	                                        //Beschränkung mögliche Nummer in der Zeile 5
	                                        FOR #i := 36 TO 44 BY 1 DO
	                                            IF #gitter[#k].nummer > 0 THEN
	                                                #gitter[#i].potenz_nummer[#gitter[#k].nummer - 1] := FALSE;
	                                            END_IF;
	                                        END_FOR;
	                                        //Beschränkung mögliche Nummer in der Säule 6
	                                        FOR #i := 5 TO 80 BY 9 DO
	                                            IF #gitter[#k].nummer > 0 THEN
	                                                #gitter[#i].potenz_nummer[#gitter[#k].nummer - 1] := FALSE;
	                                            END_IF;
	                                        END_FOR;
	                                        //Beschränkung mögliche Nummer in dem Viereck 5
	                                        #initial := 30;
	                                        #länge := 32;
	                                        FOR #m := 0 TO 2 BY 1 DO
	                                            FOR #i := #initial TO #länge BY 1 DO
	                                                IF #gitter[#k].nummer > 0 THEN
	                                                    #gitter[#i].potenz_nummer[#gitter[#k].nummer - 1] := FALSE;
	                                                END_IF;
	                                            END_FOR;
	                                            IF #m < 2 THEN
	                                                #initial := #initial + 9;
	                                                #länge := #länge + 9;
	                                            END_IF;
	                                        END_FOR;
	                                    END_REGION
	                                    //Feldchen 43
	                                42:
	                                    REGION Feldchen 43
	                                        //Beschränkung mögliche Nummer in der Zeile 5
	                                        FOR #i := 36 TO 44 BY 1 DO
	                                            IF #gitter[#k].nummer > 0 THEN
	                                                #gitter[#i].potenz_nummer[#gitter[#k].nummer - 1] := FALSE;
	                                            END_IF;
	                                        END_FOR;
	                                        //Beschränkung mögliche Nummer in der Säule 7
	                                        FOR #i := 6 TO 80 BY 9 DO
	                                            IF #gitter[#k].nummer > 0 THEN
	                                                #gitter[#i].potenz_nummer[#gitter[#k].nummer - 1] := FALSE;
	                                            END_IF;
	                                        END_FOR;
	                                        //Beschränkung mögliche Nummer in dem Viereck 6
	                                        #initial := 33;
	                                        #länge := 35;
	                                        FOR #m := 0 TO 2 BY 1 DO
	                                            FOR #i := #initial TO #länge BY 1 DO
	                                                IF #gitter[#k].nummer > 0 THEN
	                                                    #gitter[#i].potenz_nummer[#gitter[#k].nummer - 1] := FALSE;
	                                                END_IF;
	                                            END_FOR;
	                                            IF #m < 2 THEN
	                                                #initial := #initial + 9;
	                                                #länge := #länge + 9;
	                                            END_IF;
	                                        END_FOR;
	                                    END_REGION
	                                    //Feldchen 44
	                                43:
	                                    REGION Feldchen 44
	                                        //Beschränkung mögliche Nummer in der Zeile 5
	                                        FOR #i := 36 TO 44 BY 1 DO
	                                            IF #gitter[#k].nummer > 0 THEN
	                                                #gitter[#i].potenz_nummer[#gitter[#k].nummer - 1] := FALSE;
	                                            END_IF;
	                                        END_FOR;
	                                        //Beschränkung mögliche Nummer in der Säule 8
	                                        FOR #i := 7 TO 80 BY 9 DO
	                                            IF #gitter[#k].nummer > 0 THEN
	                                                #gitter[#i].potenz_nummer[#gitter[#k].nummer - 1] := FALSE;
	                                            END_IF;
	                                        END_FOR;
	                                        //Beschränkung mögliche Nummer in dem Viereck 6
	                                        #initial := 33;
	                                        #länge := 35;
	                                        FOR #m := 0 TO 2 BY 1 DO
	                                            FOR #i := #initial TO #länge BY 1 DO
	                                                IF #gitter[#k].nummer > 0 THEN
	                                                    #gitter[#i].potenz_nummer[#gitter[#k].nummer - 1] := FALSE;
	                                                END_IF;
	                                            END_FOR;
	                                            IF #m < 2 THEN
	                                                #initial := #initial + 9;
	                                                #länge := #länge + 9;
	                                            END_IF;
	                                        END_FOR;
	                                    END_REGION
	                                    //Feldchen 45
	                                44:
	                                    REGION Feldchen 45
	                                        //Beschränkung mögliche Nummer in der Zeile 5
	                                        FOR #i := 36 TO 44 BY 1 DO
	                                            IF #gitter[#k].nummer > 0 THEN
	                                                #gitter[#i].potenz_nummer[#gitter[#k].nummer - 1] := FALSE;
	                                            END_IF;
	                                        END_FOR;
	                                        //Beschränkung mögliche Nummer in der Säule 9
	                                        FOR #i := 8 TO 80 BY 9 DO
	                                            IF #gitter[#k].nummer > 0 THEN
	                                                #gitter[#i].potenz_nummer[#gitter[#k].nummer - 1] := FALSE;
	                                            END_IF;
	                                        END_FOR;
	                                        //Beschränkung mögliche Nummer in dem Viereck 6
	                                        #initial := 33;
	                                        #länge := 35;
	                                        FOR #m := 0 TO 2 BY 1 DO
	                                            FOR #i := #initial TO #länge BY 1 DO
	                                                IF #gitter[#k].nummer > 0 THEN
	                                                    #gitter[#i].potenz_nummer[#gitter[#k].nummer - 1] := FALSE;
	                                                END_IF;
	                                            END_FOR;
	                                            IF #m < 2 THEN
	                                                #initial := #initial + 9;
	                                                #länge := #länge + 9;
	                                            END_IF;
	                                        END_FOR;
	                                    END_REGION
	                                    //Feldchen 46
	                                45:
	                                    REGION Feldchen 46
	                                        //Beschränkung mögliche Nummer in der Zeile 6
	                                        FOR #i := 45 TO 53 BY 1 DO
	                                            IF #gitter[#k].nummer > 0 THEN
	                                                #gitter[#i].potenz_nummer[#gitter[#k].nummer - 1] := FALSE;
	                                            END_IF;
	                                        END_FOR;
	                                        //Beschränkung mögliche Nummer in der Säule 1
	                                        FOR #i := 0 TO 80 BY 9 DO
	                                            IF #gitter[#k].nummer > 0 THEN
	                                                #gitter[#i].potenz_nummer[#gitter[#k].nummer - 1] := FALSE;
	                                            END_IF;
	                                        END_FOR;
	                                        //Beschränkung mögliche Nummer in dem Viereck 4
	                                        #initial := 27;
	                                        #länge := 29;
	                                        FOR #m := 0 TO 2 BY 1 DO
	                                            FOR #i := #initial TO #länge BY 1 DO
	                                                IF #gitter[#k].nummer > 0 THEN
	                                                    #gitter[#i].potenz_nummer[#gitter[#k].nummer - 1] := FALSE;
	                                                END_IF;
	                                            END_FOR;
	                                            IF #m < 2 THEN
	                                                #initial := #initial + 9;
	                                                #länge := #länge + 9;
	                                            END_IF;
	                                        END_FOR;
	                                    END_REGION
	                                    //Feldchen 47
	                                46:
	                                    REGION Feldchen 47
	                                        //Beschränkung mögliche Nummer in der Zeile 6
	                                        FOR #i := 45 TO 53 BY 1 DO
	                                            IF #gitter[#k].nummer > 0 THEN
	                                                #gitter[#i].potenz_nummer[#gitter[#k].nummer - 1] := FALSE;
	                                            END_IF;
	                                        END_FOR;
	                                        //Beschränkung mögliche Nummer in der Säule 2
	                                        FOR #i := 1 TO 80 BY 9 DO
	                                            IF #gitter[#k].nummer > 0 THEN
	                                                #gitter[#i].potenz_nummer[#gitter[#k].nummer - 1] := FALSE;
	                                            END_IF;
	                                        END_FOR;
	                                        //Beschränkung mögliche Nummer in dem Viereck 4
	                                        #initial := 27;
	                                        #länge := 29;
	                                        FOR #m := 0 TO 2 BY 1 DO
	                                            FOR #i := #initial TO #länge BY 1 DO
	                                                IF #gitter[#k].nummer > 0 THEN
	                                                    #gitter[#i].potenz_nummer[#gitter[#k].nummer - 1] := FALSE;
	                                                END_IF;
	                                            END_FOR;
	                                            IF #m < 2 THEN
	                                                #initial := #initial + 9;
	                                                #länge := #länge + 9;
	                                            END_IF;
	                                        END_FOR;
	                                    END_REGION
	                                    //Feldchen 48
	                                47:
	                                    REGION Feldchen 48
	                                        //Beschränkung mögliche Nummer in der Zeile 6
	                                        FOR #i := 45 TO 53 BY 1 DO
	                                            IF #gitter[#k].nummer > 0 THEN
	                                                #gitter[#i].potenz_nummer[#gitter[#k].nummer - 1] := FALSE;
	                                            END_IF;
	                                        END_FOR;
	                                        //Beschränkung mögliche Nummer in der Säule 3
	                                        FOR #i := 2 TO 80 BY 9 DO
	                                            IF #gitter[#k].nummer > 0 THEN
	                                                #gitter[#i].potenz_nummer[#gitter[#k].nummer - 1] := FALSE;
	                                            END_IF;
	                                        END_FOR;
	                                        //Beschränkung mögliche Nummer in dem Viereck 4
	                                        #initial := 27;
	                                        #länge := 29;
	                                        FOR #m := 0 TO 2 BY 1 DO
	                                            FOR #i := #initial TO #länge BY 1 DO
	                                                IF #gitter[#k].nummer > 0 THEN
	                                                    #gitter[#i].potenz_nummer[#gitter[#k].nummer - 1] := FALSE;
	                                                END_IF;
	                                            END_FOR;
	                                            IF #m < 2 THEN
	                                                #initial := #initial + 9;
	                                                #länge := #länge + 9;
	                                            END_IF;
	                                        END_FOR;
	                                    END_REGION
	                                    //Feldchen 49
	                                48:
	                                    REGION Feldchen 49
	                                        //Beschränkung mögliche Nummer in der Zeile 6
	                                        FOR #i := 45 TO 53 BY 1 DO
	                                            IF #gitter[#k].nummer > 0 THEN
	                                                #gitter[#i].potenz_nummer[#gitter[#k].nummer - 1] := FALSE;
	                                            END_IF;
	                                        END_FOR;
	                                        //Beschränkung mögliche Nummer in der Säule 4
	                                        FOR #i := 3 TO 80 BY 9 DO
	                                            IF #gitter[#k].nummer > 0 THEN
	                                                #gitter[#i].potenz_nummer[#gitter[#k].nummer - 1] := FALSE;
	                                            END_IF;
	                                        END_FOR;
	                                        //Beschränkung mögliche Nummer in dem Viereck 5
	                                        #initial := 30;
	                                        #länge := 32;
	                                        FOR #m := 0 TO 2 BY 1 DO
	                                            FOR #i := #initial TO #länge BY 1 DO
	                                                IF #gitter[#k].nummer > 0 THEN
	                                                    #gitter[#i].potenz_nummer[#gitter[#k].nummer - 1] := FALSE;
	                                                END_IF;
	                                            END_FOR;
	                                            IF #m < 2 THEN
	                                                #initial := #initial + 9;
	                                                #länge := #länge + 9;
	                                            END_IF;
	                                        END_FOR;
	                                    END_REGION
	                                    //Feldchen 50
	                                49:
	                                    REGION Feldchen 50
	                                        //Beschränkung mögliche Nummer in der Zeile 6
	                                        FOR #i := 45 TO 53 BY 1 DO
	                                            IF #gitter[#k].nummer > 0 THEN
	                                                #gitter[#i].potenz_nummer[#gitter[#k].nummer - 1] := FALSE;
	                                            END_IF;
	                                        END_FOR;
	                                        //Beschränkung mögliche Nummer in der Säule 5
	                                        FOR #i := 4 TO 80 BY 9 DO
	                                            IF #gitter[#k].nummer > 0 THEN
	                                                #gitter[#i].potenz_nummer[#gitter[#k].nummer - 1] := FALSE;
	                                            END_IF;
	                                        END_FOR;
	                                        //Beschränkung mögliche Nummer in dem Viereck 5
	                                        #initial := 30;
	                                        #länge := 32;
	                                        FOR #m := 0 TO 2 BY 1 DO
	                                            FOR #i := #initial TO #länge BY 1 DO
	                                                IF #gitter[#k].nummer > 0 THEN
	                                                    #gitter[#i].potenz_nummer[#gitter[#k].nummer - 1] := FALSE;
	                                                END_IF;
	                                            END_FOR;
	                                            IF #m < 2 THEN
	                                                #initial := #initial + 9;
	                                                #länge := #länge + 9;
	                                            END_IF;
	                                        END_FOR;
	                                    END_REGION
	                                    //Feldchen 51
	                                50:
	                                    REGION Feldchen 51
	                                        //Beschränkung mögliche Nummer in der Zeile 6
	                                        FOR #i := 45 TO 53 BY 1 DO
	                                            IF #gitter[#k].nummer > 0 THEN
	                                                #gitter[#i].potenz_nummer[#gitter[#k].nummer - 1] := FALSE;
	                                            END_IF;
	                                        END_FOR;
	                                        //Beschränkung mögliche Nummer in der Säule 6
	                                        FOR #i := 5 TO 80 BY 9 DO
	                                            IF #gitter[#k].nummer > 0 THEN
	                                                #gitter[#i].potenz_nummer[#gitter[#k].nummer - 1] := FALSE;
	                                            END_IF;
	                                        END_FOR;
	                                        //Beschränkung mögliche Nummer in dem Viereck 5
	                                        #initial := 30;
	                                        #länge := 32;
	                                        FOR #m := 0 TO 2 BY 1 DO
	                                            FOR #i := #initial TO #länge BY 1 DO
	                                                IF #gitter[#k].nummer > 0 THEN
	                                                    #gitter[#i].potenz_nummer[#gitter[#k].nummer - 1] := FALSE;
	                                                END_IF;
	                                            END_FOR;
	                                            IF #m < 2 THEN
	                                                #initial := #initial + 9;
	                                                #länge := #länge + 9;
	                                            END_IF;
	                                        END_FOR;
	                                    END_REGION
	                                    //Feldchen 52
	                                51:
	                                    REGION Feldchen 52
	                                        //Beschränkung mögliche Nummer in der Zeile 6
	                                        FOR #i := 45 TO 53 BY 1 DO
	                                            IF #gitter[#k].nummer > 0 THEN
	                                                #gitter[#i].potenz_nummer[#gitter[#k].nummer - 1] := FALSE;
	                                            END_IF;
	                                        END_FOR;
	                                        //Beschränkung mögliche Nummer in der Säule 7
	                                        FOR #i := 6 TO 80 BY 9 DO
	                                            IF #gitter[#k].nummer > 0 THEN
	                                                #gitter[#i].potenz_nummer[#gitter[#k].nummer - 1] := FALSE;
	                                            END_IF;
	                                        END_FOR;
	                                        //Beschränkung mögliche Nummer in dem Viereck 6
	                                        #initial := 33;
	                                        #länge := 35;
	                                        FOR #m := 0 TO 2 BY 1 DO
	                                            FOR #i := #initial TO #länge BY 1 DO
	                                                IF #gitter[#k].nummer > 0 THEN
	                                                    #gitter[#i].potenz_nummer[#gitter[#k].nummer - 1] := FALSE;
	                                                END_IF;
	                                            END_FOR;
	                                            IF #m < 2 THEN
	                                                #initial := #initial + 9;
	                                                #länge := #länge + 9;
	                                            END_IF;
	                                        END_FOR;
	                                    END_REGION
	                                    //Feldchen 53
	                                52:
	                                    REGION Feldchen 53
	                                        //Beschränkung mögliche Nummer in der Zeile 6
	                                        FOR #i := 45 TO 53 BY 1 DO
	                                            IF #gitter[#k].nummer > 0 THEN
	                                                #gitter[#i].potenz_nummer[#gitter[#k].nummer - 1] := FALSE;
	                                            END_IF;
	                                        END_FOR;
	                                        //Beschränkung mögliche Nummer in der Säule 8
	                                        FOR #i := 7 TO 80 BY 9 DO
	                                            IF #gitter[#k].nummer > 0 THEN
	                                                #gitter[#i].potenz_nummer[#gitter[#k].nummer - 1] := FALSE;
	                                            END_IF;
	                                        END_FOR;
	                                        //Beschränkung mögliche Nummer in dem Viereck 6
	                                        #initial := 33;
	                                        #länge := 35;
	                                        FOR #m := 0 TO 2 BY 1 DO
	                                            FOR #i := #initial TO #länge BY 1 DO
	                                                IF #gitter[#k].nummer > 0 THEN
	                                                    #gitter[#i].potenz_nummer[#gitter[#k].nummer - 1] := FALSE;
	                                                END_IF;
	                                            END_FOR;
	                                            IF #m < 2 THEN
	                                                #initial := #initial + 9;
	                                                #länge := #länge + 9;
	                                            END_IF;
	                                        END_FOR;
	                                    END_REGION
	                                    //Feldchen 54
	                                53:
	                                    REGION Feldchen 54
	                                        //Beschränkung mögliche Nummer in der Zeile 6
	                                        FOR #i := 45 TO 53 BY 1 DO
	                                            IF #gitter[#k].nummer > 0 THEN
	                                                #gitter[#i].potenz_nummer[#gitter[#k].nummer - 1] := FALSE;
	                                            END_IF;
	                                        END_FOR;
	                                        //Beschränkung mögliche Nummer in der Säule 9
	                                        FOR #i := 8 TO 80 BY 9 DO
	                                            IF #gitter[#k].nummer > 0 THEN
	                                                #gitter[#i].potenz_nummer[#gitter[#k].nummer - 1] := FALSE;
	                                            END_IF;
	                                        END_FOR;
	                                        //Beschränkung mögliche Nummer in dem Viereck 6
	                                        #initial := 33;
	                                        #länge := 35;
	                                        FOR #m := 0 TO 2 BY 1 DO
	                                            FOR #i := #initial TO #länge BY 1 DO
	                                                IF #gitter[#k].nummer > 0 THEN
	                                                    #gitter[#i].potenz_nummer[#gitter[#k].nummer - 1] := FALSE;
	                                                END_IF;
	                                            END_FOR;
	                                            IF #m < 2 THEN
	                                                #initial := #initial + 9;
	                                                #länge := #länge + 9;
	                                            END_IF;
	                                        END_FOR;
	                                    END_REGION
	                                    //Feldchen 55
	                                54:
	                                    REGION Feldchen 55
	                                        //Beschränkung mögliche Nummer in der Zeile 7
	                                        FOR #i := 54 TO 62 BY 1 DO
	                                            IF #gitter[#k].nummer > 0 THEN
	                                                #gitter[#i].potenz_nummer[#gitter[#k].nummer - 1] := FALSE;
	                                            END_IF;
	                                        END_FOR;
	                                        //Beschränkung mögliche Nummer in der Säule 1
	                                        FOR #i := 0 TO 80 BY 9 DO
	                                            IF #gitter[#k].nummer > 0 THEN
	                                                #gitter[#i].potenz_nummer[#gitter[#k].nummer - 1] := FALSE;
	                                            END_IF;
	                                        END_FOR;
	                                        //Beschränkung mögliche Nummer in dem Viereck 7
	                                        #initial := 54;
	                                        #länge := 56;
	                                        FOR #m := 0 TO 2 BY 1 DO
	                                            FOR #i := #initial TO #länge BY 1 DO
	                                                IF #gitter[#k].nummer > 0 THEN
	                                                    #gitter[#i].potenz_nummer[#gitter[#k].nummer - 1] := FALSE;
	                                                END_IF;
	                                            END_FOR;
	                                            IF #m < 2 THEN
	                                                #initial := #initial + 9;
	                                                #länge := #länge + 9;
	                                            END_IF;
	                                        END_FOR;
	                                    END_REGION
	                                    //Feldchen 56
	                                55:
	                                    REGION Feldchen 56
	                                        //Beschränkung mögliche Nummer in der Zeile 7
	                                        FOR #i := 54 TO 62 BY 1 DO
	                                            IF #gitter[#k].nummer > 0 THEN
	                                                #gitter[#i].potenz_nummer[#gitter[#k].nummer - 1] := FALSE;
	                                            END_IF;
	                                        END_FOR;
	                                        //Beschränkung mögliche Nummer in der Säule 2
	                                        FOR #i := 1 TO 80 BY 9 DO
	                                            IF #gitter[#k].nummer > 0 THEN
	                                                #gitter[#i].potenz_nummer[#gitter[#k].nummer - 1] := FALSE;
	                                            END_IF;
	                                        END_FOR;
	                                        //Beschränkung mögliche Nummer in dem Viereck 7
	                                        #initial := 54;
	                                        #länge := 56;
	                                        FOR #m := 0 TO 2 BY 1 DO
	                                            FOR #i := #initial TO #länge BY 1 DO
	                                                IF #gitter[#k].nummer > 0 THEN
	                                                    #gitter[#i].potenz_nummer[#gitter[#k].nummer - 1] := FALSE;
	                                                END_IF;
	                                            END_FOR;
	                                            IF #m < 2 THEN
	                                                #initial := #initial + 9;
	                                                #länge := #länge + 9;
	                                            END_IF;
	                                        END_FOR;
	                                    END_REGION
	                                    //Feldchen 57
	                                56:
	                                    REGION Feldchen 57
	                                        //Beschränkung mögliche Nummer in der Zeile 7
	                                        FOR #i := 54 TO 62 BY 1 DO
	                                            IF #gitter[#k].nummer > 0 THEN
	                                                #gitter[#i].potenz_nummer[#gitter[#k].nummer - 1] := FALSE;
	                                            END_IF;
	                                        END_FOR;
	                                        //Beschränkung mögliche Nummer in der Säule 3
	                                        FOR #i := 2 TO 80 BY 9 DO
	                                            IF #gitter[#k].nummer > 0 THEN
	                                                #gitter[#i].potenz_nummer[#gitter[#k].nummer - 1] := FALSE;
	                                            END_IF;
	                                        END_FOR;
	                                        //Beschränkung mögliche Nummer in dem Viereck 7
	                                        #initial := 54;
	                                        #länge := 56;
	                                        FOR #m := 0 TO 2 BY 1 DO
	                                            FOR #i := #initial TO #länge BY 1 DO
	                                                IF #gitter[#k].nummer > 0 THEN
	                                                    #gitter[#i].potenz_nummer[#gitter[#k].nummer - 1] := FALSE;
	                                                END_IF;
	                                            END_FOR;
	                                            IF #m < 2 THEN
	                                                #initial := #initial + 9;
	                                                #länge := #länge + 9;
	                                            END_IF;
	                                        END_FOR;
	                                    END_REGION //Feldchen 57
	                                    //Feldchen 58
	                                57:
	                                    REGION Feldchen 58
	                                        //Beschränkung mögliche Nummer in der Zeile 7
	                                        FOR #i := 54 TO 62 BY 1 DO
	                                            IF #gitter[#k].nummer > 0 THEN
	                                                #gitter[#i].potenz_nummer[#gitter[#k].nummer - 1] := FALSE;
	                                            END_IF;
	                                        END_FOR;
	                                        //Beschränkung mögliche Nummer in der Säule 4
	                                        FOR #i := 3 TO 80 BY 9 DO
	                                            IF #gitter[#k].nummer > 0 THEN
	                                                #gitter[#i].potenz_nummer[#gitter[#k].nummer - 1] := FALSE;
	                                            END_IF;
	                                        END_FOR;
	                                        //Beschränkung mögliche Nummer in dem Viereck 8
	                                        #initial := 57;
	                                        #länge := 59;
	                                        FOR #m := 0 TO 2 BY 1 DO
	                                            FOR #i := #initial TO #länge BY 1 DO
	                                                IF #gitter[#k].nummer > 0 THEN
	                                                    #gitter[#i].potenz_nummer[#gitter[#k].nummer - 1] := FALSE;
	                                                END_IF;
	                                            END_FOR;
	                                            IF #m < 2 THEN
	                                                #initial := #initial + 9;
	                                                #länge := #länge + 9;
	                                            END_IF;
	                                        END_FOR;
	                                    END_REGION
	                                    //Feldchen 59
	                                58:
	                                    REGION Feldchen 59
	                                        //Beschränkung mögliche Nummer in der Zeile 7
	                                        FOR #i := 54 TO 62 BY 1 DO
	                                            IF #gitter[#k].nummer > 0 THEN
	                                                #gitter[#i].potenz_nummer[#gitter[#k].nummer - 1] := FALSE;
	                                            END_IF;
	                                        END_FOR;
	                                        //Beschränkung mögliche Nummer in der Säule 5
	                                        FOR #i := 4 TO 80 BY 9 DO
	                                            IF #gitter[#k].nummer > 0 THEN
	                                                #gitter[#i].potenz_nummer[#gitter[#k].nummer - 1] := FALSE;
	                                            END_IF;
	                                        END_FOR;
	                                        //Beschränkung mögliche Nummer in dem Viereck 8
	                                        #initial := 57;
	                                        #länge := 59;
	                                        FOR #m := 0 TO 2 BY 1 DO
	                                            FOR #i := #initial TO #länge BY 1 DO
	                                                IF #gitter[#k].nummer > 0 THEN
	                                                    #gitter[#i].potenz_nummer[#gitter[#k].nummer - 1] := FALSE;
	                                                END_IF;
	                                            END_FOR;
	                                            IF #m < 2 THEN
	                                                #initial := #initial + 9;
	                                                #länge := #länge + 9;
	                                            END_IF;
	                                        END_FOR;
	                                    END_REGION
	                                    //Feldchen 60
	                                59:
	                                    REGION Feldchen 60
	                                        //Beschränkung mögliche Nummer in der Zeile 7
	                                        FOR #i := 54 TO 62 BY 1 DO
	                                            IF #gitter[#k].nummer > 0 THEN
	                                                #gitter[#i].potenz_nummer[#gitter[#k].nummer - 1] := FALSE;
	                                            END_IF;
	                                        END_FOR;
	                                        //Beschränkung mögliche Nummer in der Säule 6
	                                        FOR #i := 5 TO 80 BY 9 DO
	                                            IF #gitter[#k].nummer > 0 THEN
	                                                #gitter[#i].potenz_nummer[#gitter[#k].nummer - 1] := FALSE;
	                                            END_IF;
	                                        END_FOR;
	                                        //Beschränkung mögliche Nummer in dem Viereck 8
	                                        #initial := 57;
	                                        #länge := 59;
	                                        FOR #m := 0 TO 2 BY 1 DO
	                                            FOR #i := #initial TO #länge BY 1 DO
	                                                IF #gitter[#k].nummer > 0 THEN
	                                                    #gitter[#i].potenz_nummer[#gitter[#k].nummer - 1] := FALSE;
	                                                END_IF;
	                                            END_FOR;
	                                            IF #m < 2 THEN
	                                                #initial := #initial + 9;
	                                                #länge := #länge + 9;
	                                            END_IF;
	                                        END_FOR;
	                                    END_REGION
	                                    //Feldchen 61
	                                60:
	                                    REGION Feldchen 61
	                                        //Beschränkung mögliche Nummer in der Zeile 7
	                                        FOR #i := 54 TO 62 BY 1 DO
	                                            IF #gitter[#k].nummer > 0 THEN
	                                                #gitter[#i].potenz_nummer[#gitter[#k].nummer - 1] := FALSE;
	                                            END_IF;
	                                        END_FOR;
	                                        //Beschränkung mögliche Nummer in der Säule 7
	                                        FOR #i := 6 TO 80 BY 9 DO
	                                            IF #gitter[#k].nummer > 0 THEN
	                                                #gitter[#i].potenz_nummer[#gitter[#k].nummer - 1] := FALSE;
	                                            END_IF;
	                                        END_FOR;
	                                        //Beschränkung mögliche Nummer in dem Viereck 9
	                                        #initial := 60;
	                                        #länge := 62;
	                                        FOR #m := 0 TO 2 BY 1 DO
	                                            FOR #i := #initial TO #länge BY 1 DO
	                                                IF #gitter[#k].nummer > 0 THEN
	                                                    #gitter[#i].potenz_nummer[#gitter[#k].nummer - 1] := FALSE;
	                                                END_IF;
	                                            END_FOR;
	                                            IF #m < 2 THEN
	                                                #initial := #initial + 9;
	                                                #länge := #länge + 9;
	                                            END_IF;
	                                        END_FOR;
	                                    END_REGION
	                                    //Feldchen 62
	                                61:
	                                    REGION Feldchen 62
	                                        //Beschränkung mögliche Nummer in der Zeile 7
	                                        FOR #i := 54 TO 62 BY 1 DO
	                                            IF #gitter[#k].nummer > 0 THEN
	                                                #gitter[#i].potenz_nummer[#gitter[#k].nummer - 1] := FALSE;
	                                            END_IF;
	                                        END_FOR;
	                                        //Beschränkung mögliche Nummer in der Säule 8
	                                        FOR #i := 7 TO 80 BY 9 DO
	                                            IF #gitter[#k].nummer > 0 THEN
	                                                #gitter[#i].potenz_nummer[#gitter[#k].nummer - 1] := FALSE;
	                                            END_IF;
	                                        END_FOR;
	                                        //Beschränkung mögliche Nummer in dem Viereck 9
	                                        #initial := 60;
	                                        #länge := 62;
	                                        FOR #m := 0 TO 2 BY 1 DO
	                                            FOR #i := #initial TO #länge BY 1 DO
	                                                IF #gitter[#k].nummer > 0 THEN
	                                                    #gitter[#i].potenz_nummer[#gitter[#k].nummer - 1] := FALSE;
	                                                END_IF;
	                                            END_FOR;
	                                            IF #m < 2 THEN
	                                                #initial := #initial + 9;
	                                                #länge := #länge + 9;
	                                            END_IF;
	                                        END_FOR;
	                                    END_REGION
	                                    //Feldchen 63
	                                62:
	                                    REGION Feldchen 63
	                                        //Beschränkung mögliche Nummer in der Zeile 7
	                                        FOR #i := 54 TO 62 BY 1 DO
	                                            IF #gitter[#k].nummer > 0 THEN
	                                                #gitter[#i].potenz_nummer[#gitter[#k].nummer - 1] := FALSE;
	                                            END_IF;
	                                        END_FOR;
	                                        //Beschränkung mögliche Nummer in der Säule 9
	                                        FOR #i := 8 TO 80 BY 9 DO
	                                            IF #gitter[#k].nummer > 0 THEN
	                                                #gitter[#i].potenz_nummer[#gitter[#k].nummer - 1] := FALSE;
	                                            END_IF;
	                                        END_FOR;
	                                        //Beschränkung mögliche Nummer in dem Viereck 9
	                                        #initial := 60;
	                                        #länge := 62;
	                                        FOR #m := 0 TO 2 BY 1 DO
	                                            FOR #i := #initial TO #länge BY 1 DO
	                                                IF #gitter[#k].nummer > 0 THEN
	                                                    #gitter[#i].potenz_nummer[#gitter[#k].nummer - 1] := FALSE;
	                                                END_IF;
	                                            END_FOR;
	                                            IF #m < 2 THEN
	                                                #initial := #initial + 9;
	                                                #länge := #länge + 9;
	                                            END_IF;
	                                        END_FOR;
	                                    END_REGION
	                                    //Feldchen 64
	                                63:
	                                    REGION Feldchen 64
	                                        //Beschränkung mögliche Nummer in der Zeile 8
	                                        FOR #i := 63 TO 71 BY 1 DO
	                                            IF #gitter[#k].nummer > 0 THEN
	                                                #gitter[#i].potenz_nummer[#gitter[#k].nummer - 1] := FALSE;
	                                            END_IF;
	                                        END_FOR;
	                                        //Beschränkung mögliche Nummer in der Säule 1
	                                        FOR #i := 0 TO 80 BY 9 DO
	                                            IF #gitter[#k].nummer > 0 THEN
	                                                #gitter[#i].potenz_nummer[#gitter[#k].nummer - 1] := FALSE;
	                                            END_IF;
	                                        END_FOR;
	                                        //Beschränkung mögliche Nummer in dem Viereck 7
	                                        #initial := 54;
	                                        #länge := 56;
	                                        FOR #m := 0 TO 2 BY 1 DO
	                                            FOR #i := #initial TO #länge BY 1 DO
	                                                IF #gitter[#k].nummer > 0 THEN
	                                                    #gitter[#i].potenz_nummer[#gitter[#k].nummer - 1] := FALSE;
	                                                END_IF;
	                                            END_FOR;
	                                            IF #m < 2 THEN
	                                                #initial := #initial + 9;
	                                                #länge := #länge + 9;
	                                            END_IF;
	                                        END_FOR;
	                                    END_REGION
	                                    //Feldchen 65
	                                64:
	                                    REGION Feldchen 65
	                                        //Beschränkung mögliche Nummer in der Zeile 8
	                                        FOR #i := 63 TO 71 BY 1 DO
	                                            IF #gitter[#k].nummer > 0 THEN
	                                                #gitter[#i].potenz_nummer[#gitter[#k].nummer - 1] := FALSE;
	                                            END_IF;
	                                        END_FOR;
	                                        //Beschränkung mögliche Nummer in der Säule 2
	                                        FOR #i := 1 TO 80 BY 9 DO
	                                            IF #gitter[#k].nummer > 0 THEN
	                                                #gitter[#i].potenz_nummer[#gitter[#k].nummer - 1] := FALSE;
	                                            END_IF;
	                                        END_FOR;
	                                        //Beschränkung mögliche Nummer in dem Viereck 7
	                                        #initial := 54;
	                                        #länge := 56;
	                                        FOR #m := 0 TO 2 BY 1 DO
	                                            FOR #i := #initial TO #länge BY 1 DO
	                                                IF #gitter[#k].nummer > 0 THEN
	                                                    #gitter[#i].potenz_nummer[#gitter[#k].nummer - 1] := FALSE;
	                                                END_IF;
	                                            END_FOR;
	                                            IF #m < 2 THEN
	                                                #initial := #initial + 9;
	                                                #länge := #länge + 9;
	                                            END_IF;
	                                        END_FOR;
	                                    END_REGION
	                                    //Feldchen 66
	                                65:
	                                    REGION Feldchen 66
	                                        //Beschränkung mögliche Nummer in der Zeile 8
	                                        FOR #i := 63 TO 71 BY 1 DO
	                                            IF #gitter[#k].nummer > 0 THEN
	                                                #gitter[#i].potenz_nummer[#gitter[#k].nummer - 1] := FALSE;
	                                            END_IF;
	                                        END_FOR;
	                                        //Beschränkung mögliche Nummer in der Säule 3
	                                        FOR #i := 2 TO 80 BY 9 DO
	                                            IF #gitter[#k].nummer > 0 THEN
	                                                #gitter[#i].potenz_nummer[#gitter[#k].nummer - 1] := FALSE;
	                                            END_IF;
	                                        END_FOR;
	                                        //Beschränkung mögliche Nummer in dem Viereck 7
	                                        #initial := 54;
	                                        #länge := 56;
	                                        FOR #m := 0 TO 2 BY 1 DO
	                                            FOR #i := #initial TO #länge BY 1 DO
	                                                IF #gitter[#k].nummer > 0 THEN
	                                                    #gitter[#i].potenz_nummer[#gitter[#k].nummer - 1] := FALSE;
	                                                END_IF;
	                                            END_FOR;
	                                            IF #m < 2 THEN
	                                                #initial := #initial + 9;
	                                                #länge := #länge + 9;
	                                            END_IF;
	                                        END_FOR;
	                                    END_REGION
	                                    //Feldchen 67
	                                66:
	                                    REGION Feldchen 67
	                                        //Beschränkung mögliche Nummer in der Zeile 8
	                                        FOR #i := 63 TO 71 BY 1 DO
	                                            IF #gitter[#k].nummer > 0 THEN
	                                                #gitter[#i].potenz_nummer[#gitter[#k].nummer - 1] := FALSE;
	                                            END_IF;
	                                        END_FOR;
	                                        //Beschränkung mögliche Nummer in der Säule 4
	                                        FOR #i := 3 TO 80 BY 9 DO
	                                            IF #gitter[#k].nummer > 0 THEN
	                                                #gitter[#i].potenz_nummer[#gitter[#k].nummer - 1] := FALSE;
	                                            END_IF;
	                                        END_FOR;
	                                        //Beschränkung mögliche Nummer in dem Viereck 8
	                                        #initial := 57;
	                                        #länge := 59;
	                                        FOR #m := 0 TO 2 BY 1 DO
	                                            FOR #i := #initial TO #länge BY 1 DO
	                                                IF #gitter[#k].nummer > 0 THEN
	                                                    #gitter[#i].potenz_nummer[#gitter[#k].nummer - 1] := FALSE;
	                                                END_IF;
	                                            END_FOR;
	                                            IF #m < 2 THEN
	                                                #initial := #initial + 9;
	                                                #länge := #länge + 9;
	                                            END_IF;
	                                        END_FOR;
	                                    END_REGION
	                                    //Feldchen 68
	                                67:
	                                    REGION Feldchen 68
	                                        //Beschränkung mögliche Nummer in der Zeile 8
	                                        FOR #i := 63 TO 71 BY 1 DO
	                                            IF #gitter[#k].nummer > 0 THEN
	                                                #gitter[#i].potenz_nummer[#gitter[#k].nummer - 1] := FALSE;
	                                            END_IF;
	                                        END_FOR;
	                                        //Beschränkung mögliche Nummer in der Säule 5
	                                        FOR #i := 4 TO 80 BY 9 DO
	                                            IF #gitter[#k].nummer > 0 THEN
	                                                #gitter[#i].potenz_nummer[#gitter[#k].nummer - 1] := FALSE;
	                                            END_IF;
	                                        END_FOR;
	                                        //Beschränkung mögliche Nummer in dem Viereck 8
	                                        #initial := 57;
	                                        #länge := 59;
	                                        FOR #m := 0 TO 2 BY 1 DO
	                                            FOR #i := #initial TO #länge BY 1 DO
	                                                IF #gitter[#k].nummer > 0 THEN
	                                                    #gitter[#i].potenz_nummer[#gitter[#k].nummer - 1] := FALSE;
	                                                END_IF;
	                                            END_FOR;
	                                            IF #m < 2 THEN
	                                                #initial := #initial + 9;
	                                                #länge := #länge + 9;
	                                            END_IF;
	                                        END_FOR;
	                                    END_REGION
	                                    //Feldchen 69
	                                68:
	                                    REGION Feldchen 69
	                                        //Beschränkung mögliche Nummer in der Zeile 8
	                                        FOR #i := 63 TO 71 BY 1 DO
	                                            IF #gitter[#k].nummer > 0 THEN
	                                                #gitter[#i].potenz_nummer[#gitter[#k].nummer - 1] := FALSE;
	                                            END_IF;
	                                        END_FOR;
	                                        //Beschränkung mögliche Nummer in der Säule 6
	                                        FOR #i := 5 TO 80 BY 9 DO
	                                            IF #gitter[#k].nummer > 0 THEN
	                                                #gitter[#i].potenz_nummer[#gitter[#k].nummer - 1] := FALSE;
	                                            END_IF;
	                                        END_FOR;
	                                        //Beschränkung mögliche Nummer in dem Viereck 8
	                                        #initial := 57;
	                                        #länge := 59;
	                                        FOR #m := 0 TO 2 BY 1 DO
	                                            FOR #i := #initial TO #länge BY 1 DO
	                                                IF #gitter[#k].nummer > 0 THEN
	                                                    #gitter[#i].potenz_nummer[#gitter[#k].nummer - 1] := FALSE;
	                                                END_IF;
	                                            END_FOR;
	                                            IF #m < 2 THEN
	                                                #initial := #initial + 9;
	                                                #länge := #länge + 9;
	                                            END_IF;
	                                        END_FOR;
	                                    END_REGION
	                                    //Feldchen 70
	                                69:
	                                    REGION Feldchen 70
	                                        //Beschränkung mögliche Nummer in der Zeile 8
	                                        FOR #i := 63 TO 71 BY 1 DO
	                                            IF #gitter[#k].nummer > 0 THEN
	                                                #gitter[#i].potenz_nummer[#gitter[#k].nummer - 1] := FALSE;
	                                            END_IF;
	                                        END_FOR;
	                                        //Beschränkung mögliche Nummer in der Säule 7
	                                        FOR #i := 6 TO 80 BY 9 DO
	                                            IF #gitter[#k].nummer > 0 THEN
	                                                #gitter[#i].potenz_nummer[#gitter[#k].nummer - 1] := FALSE;
	                                            END_IF;
	                                        END_FOR;
	                                        //Beschränkung mögliche Nummer in dem Viereck 9
	                                        #initial := 60;
	                                        #länge := 62;
	                                        FOR #m := 0 TO 2 BY 1 DO
	                                            FOR #i := #initial TO #länge BY 1 DO
	                                                IF #gitter[#k].nummer > 0 THEN
	                                                    #gitter[#i].potenz_nummer[#gitter[#k].nummer - 1] := FALSE;
	                                                END_IF;
	                                            END_FOR;
	                                            IF #m < 2 THEN
	                                                #initial := #initial + 9;
	                                                #länge := #länge + 9;
	                                            END_IF;
	                                        END_FOR;
	                                    END_REGION
	                                    //Feldchen 71
	                                70:
	                                    REGION Feldchen 71
	                                        //Beschränkung mögliche Nummer in der Zeile 8
	                                        FOR #i := 63 TO 71 BY 1 DO
	                                            IF #gitter[#k].nummer > 0 THEN
	                                                #gitter[#i].potenz_nummer[#gitter[#k].nummer - 1] := FALSE;
	                                            END_IF;
	                                        END_FOR;
	                                        //Beschränkung mögliche Nummer in der Säule 8
	                                        FOR #i := 7 TO 80 BY 9 DO
	                                            IF #gitter[#k].nummer > 0 THEN
	                                                #gitter[#i].potenz_nummer[#gitter[#k].nummer - 1] := FALSE;
	                                            END_IF;
	                                        END_FOR;
	                                        //Beschränkung mögliche Nummer in dem Viereck 9
	                                        #initial := 60;
	                                        #länge := 62;
	                                        FOR #m := 0 TO 2 BY 1 DO
	                                            FOR #i := #initial TO #länge BY 1 DO
	                                                IF #gitter[#k].nummer > 0 THEN
	                                                    #gitter[#i].potenz_nummer[#gitter[#k].nummer - 1] := FALSE;
	                                                END_IF;
	                                            END_FOR;
	                                            IF #m < 2 THEN
	                                                #initial := #initial + 9;
	                                                #länge := #länge + 9;
	                                            END_IF;
	                                        END_FOR;
	                                    END_REGION
	                                    //Feldchen 72
	                                71:
	                                    REGION Feldchen 72
	                                        //Beschränkung mögliche Nummer in der Zeile 8
	                                        FOR #i := 63 TO 71 BY 1 DO
	                                            IF #gitter[#k].nummer > 0 THEN
	                                                #gitter[#i].potenz_nummer[#gitter[#k].nummer - 1] := FALSE;
	                                            END_IF;
	                                        END_FOR;
	                                        //Beschränkung mögliche Nummer in der Säule 9
	                                        FOR #i := 8 TO 80 BY 9 DO
	                                            IF #gitter[#k].nummer > 0 THEN
	                                                #gitter[#i].potenz_nummer[#gitter[#k].nummer - 1] := FALSE;
	                                            END_IF;
	                                        END_FOR;
	                                        //Beschränkung mögliche Nummer in dem Viereck 9
	                                        #initial := 60;
	                                        #länge := 62;
	                                        FOR #m := 0 TO 2 BY 1 DO
	                                            FOR #i := #initial TO #länge BY 1 DO
	                                                IF #gitter[#k].nummer > 0 THEN
	                                                    #gitter[#i].potenz_nummer[#gitter[#k].nummer - 1] := FALSE;
	                                                END_IF;
	                                            END_FOR;
	                                            IF #m < 2 THEN
	                                                #initial := #initial + 9;
	                                                #länge := #länge + 9;
	                                            END_IF;
	                                        END_FOR;
	                                    END_REGION
	                                    //Feldchen 73
	                                72:
	                                    REGION Feldchen 73
	                                        //Beschränkung mögliche Nummer in der Zeile 9
	                                        FOR #i := 72 TO 80 BY 1 DO
	                                            IF #gitter[#k].nummer > 0 THEN
	                                                #gitter[#i].potenz_nummer[#gitter[#k].nummer - 1] := FALSE;
	                                            END_IF;
	                                        END_FOR;
	                                        //Beschränkung mögliche Nummer in der Säule 1
	                                        FOR #i := 0 TO 80 BY 9 DO
	                                            IF #gitter[#k].nummer > 0 THEN
	                                                #gitter[#i].potenz_nummer[#gitter[#k].nummer - 1] := FALSE;
	                                            END_IF;
	                                        END_FOR;
	                                        //Beschränkung mögliche Nummer in dem Viereck 7
	                                        #initial := 54;
	                                        #länge := 56;
	                                        FOR #m := 0 TO 2 BY 1 DO
	                                            FOR #i := #initial TO #länge BY 1 DO
	                                                IF #gitter[#k].nummer > 0 THEN
	                                                    #gitter[#i].potenz_nummer[#gitter[#k].nummer - 1] := FALSE;
	                                                END_IF;
	                                            END_FOR;
	                                            IF #m < 2 THEN
	                                                #initial := #initial + 9;
	                                                #länge := #länge + 9;
	                                            END_IF;
	                                        END_FOR;
	                                    END_REGION
	                                    //Feldchen 74
	                                73:
	                                    REGION Feldchen 74
	                                        //Beschränkung mögliche Nummer in der Zeile 9
	                                        FOR #i := 72 TO 80 BY 1 DO
	                                            IF #gitter[#k].nummer > 0 THEN
	                                                #gitter[#i].potenz_nummer[#gitter[#k].nummer - 1] := FALSE;
	                                            END_IF;
	                                        END_FOR;
	                                        //Beschränkung mögliche Nummer in der Säule 2
	                                        FOR #i := 1 TO 80 BY 9 DO
	                                            IF #gitter[#k].nummer > 0 THEN
	                                                #gitter[#i].potenz_nummer[#gitter[#k].nummer - 1] := FALSE;
	                                            END_IF;
	                                        END_FOR;
	                                        //Beschränkung mögliche Nummer in dem Viereck 7
	                                        #initial := 54;
	                                        #länge := 56;
	                                        FOR #m := 0 TO 2 BY 1 DO
	                                            FOR #i := #initial TO #länge BY 1 DO
	                                                IF #gitter[#k].nummer > 0 THEN
	                                                    #gitter[#i].potenz_nummer[#gitter[#k].nummer - 1] := FALSE;
	                                                END_IF;
	                                            END_FOR;
	                                            IF #m < 2 THEN
	                                                #initial := #initial + 9;
	                                                #länge := #länge + 9;
	                                            END_IF;
	                                        END_FOR;
	                                    END_REGION
	                                    //Feldchen 75
	                                74:
	                                    REGION Feldchen 75
	                                        //Beschränkung mögliche Nummer in der Zeile 9
	                                        FOR #i := 72 TO 80 BY 1 DO
	                                            IF #gitter[#k].nummer > 0 THEN
	                                                #gitter[#i].potenz_nummer[#gitter[#k].nummer - 1] := FALSE;
	                                            END_IF;
	                                        END_FOR;
	                                        //Beschränkung mögliche Nummer in der Säule 3
	                                        FOR #i := 2 TO 80 BY 9 DO
	                                            IF #gitter[#k].nummer > 0 THEN
	                                                #gitter[#i].potenz_nummer[#gitter[#k].nummer - 1] := FALSE;
	                                            END_IF;
	                                        END_FOR;
	                                        //Beschränkung mögliche Nummer in dem Viereck 7
	                                        #initial := 54;
	                                        #länge := 56;
	                                        FOR #m := 0 TO 2 BY 1 DO
	                                            FOR #i := #initial TO #länge BY 1 DO
	                                                IF #gitter[#k].nummer > 0 THEN
	                                                    #gitter[#i].potenz_nummer[#gitter[#k].nummer - 1] := FALSE;
	                                                END_IF;
	                                            END_FOR;
	                                            IF #m < 2 THEN
	                                                #initial := #initial + 9;
	                                                #länge := #länge + 9;
	                                            END_IF;
	                                        END_FOR;
	                                    END_REGION
	                                    //Feldchen 76
	                                75:
	                                    REGION Feldchen 76
	                                        //Beschränkung mögliche Nummer in der Zeile 9
	                                        FOR #i := 72 TO 80 BY 1 DO
	                                            IF #gitter[#k].nummer > 0 THEN
	                                                #gitter[#i].potenz_nummer[#gitter[#k].nummer - 1] := FALSE;
	                                            END_IF;
	                                        END_FOR;
	                                        //Beschränkung mögliche Nummer in der Säule 4
	                                        FOR #i := 3 TO 80 BY 9 DO
	                                            IF #gitter[#k].nummer > 0 THEN
	                                                #gitter[#i].potenz_nummer[#gitter[#k].nummer - 1] := FALSE;
	                                            END_IF;
	                                        END_FOR;
	                                        //Beschränkung mögliche Nummer in dem Viereck 8
	                                        #initial := 57;
	                                        #länge := 59;
	                                        FOR #m := 0 TO 2 BY 1 DO
	                                            FOR #i := #initial TO #länge BY 1 DO
	                                                IF #gitter[#k].nummer > 0 THEN
	                                                    #gitter[#i].potenz_nummer[#gitter[#k].nummer - 1] := FALSE;
	                                                END_IF;
	                                            END_FOR;
	                                            IF #m < 2 THEN
	                                                #initial := #initial + 9;
	                                                #länge := #länge + 9;
	                                            END_IF;
	                                        END_FOR;
	                                    END_REGION
	                                    //Feldchen 77
	                                76:
	                                    REGION Feldchen 77
	                                        //Beschränkung mögliche Nummer in der Zeile 9
	                                        FOR #i := 72 TO 80 BY 1 DO
	                                            IF #gitter[#k].nummer > 0 THEN
	                                                #gitter[#i].potenz_nummer[#gitter[#k].nummer - 1] := FALSE;
	                                            END_IF;
	                                        END_FOR;
	                                        //Beschränkung mögliche Nummer in der Säule 5
	                                        FOR #i := 4 TO 80 BY 9 DO
	                                            IF #gitter[#k].nummer > 0 THEN
	                                                #gitter[#i].potenz_nummer[#gitter[#k].nummer - 1] := FALSE;
	                                            END_IF;
	                                        END_FOR;
	                                        //Beschränkung mögliche Nummer in dem Viereck 8
	                                        #initial := 57;
	                                        #länge := 59;
	                                        FOR #m := 0 TO 2 BY 1 DO
	                                            FOR #i := #initial TO #länge BY 1 DO
	                                                IF #gitter[#k].nummer > 0 THEN
	                                                    #gitter[#i].potenz_nummer[#gitter[#k].nummer - 1] := FALSE;
	                                                END_IF;
	                                            END_FOR;
	                                            IF #m < 2 THEN
	                                                #initial := #initial + 9;
	                                                #länge := #länge + 9;
	                                            END_IF;
	                                        END_FOR;
	                                    END_REGION
	                                    //Feldchen 78
	                                77:
	                                    REGION Feldchen 78
	                                        //Beschränkung mögliche Nummer in der Zeile 9
	                                        FOR #i := 72 TO 80 BY 1 DO
	                                            IF #gitter[#k].nummer > 0 THEN
	                                                #gitter[#i].potenz_nummer[#gitter[#k].nummer - 1] := FALSE;
	                                            END_IF;
	                                        END_FOR;
	                                        //Beschränkung mögliche Nummer in der Säule 6
	                                        FOR #i := 5 TO 80 BY 9 DO
	                                            IF #gitter[#k].nummer > 0 THEN
	                                                #gitter[#i].potenz_nummer[#gitter[#k].nummer - 1] := FALSE;
	                                            END_IF;
	                                        END_FOR;
	                                        //Beschränkung mögliche Nummer in dem Viereck 8
	                                        #initial := 57;
	                                        #länge := 59;
	                                        FOR #m := 0 TO 2 BY 1 DO
	                                            FOR #i := #initial TO #länge BY 1 DO
	                                                IF #gitter[#k].nummer > 0 THEN
	                                                    #gitter[#i].potenz_nummer[#gitter[#k].nummer - 1] := FALSE;
	                                                END_IF;
	                                            END_FOR;
	                                            IF #m < 2 THEN
	                                                #initial := #initial + 9;
	                                                #länge := #länge + 9;
	                                            END_IF;
	                                        END_FOR;
	                                    END_REGION
	                                    //Feldchen 79
	                                78:
	                                    REGION Feldchen 79
	                                        //Beschränkung mögliche Nummer in der Zeile 9
	                                        FOR #i := 72 TO 80 BY 1 DO
	                                            IF #gitter[#k].nummer > 0 THEN
	                                                #gitter[#i].potenz_nummer[#gitter[#k].nummer - 1] := FALSE;
	                                            END_IF;
	                                        END_FOR;
	                                        //Beschränkung mögliche Nummer in der Säule 7
	                                        FOR #i := 6 TO 80 BY 9 DO
	                                            IF #gitter[#k].nummer > 0 THEN
	                                                #gitter[#i].potenz_nummer[#gitter[#k].nummer - 1] := FALSE;
	                                            END_IF;
	                                        END_FOR;
	                                        //Beschränkung mögliche Nummer in dem Viereck 9
	                                        #initial := 60;
	                                        #länge := 62;
	                                        FOR #m := 0 TO 2 BY 1 DO
	                                            FOR #i := #initial TO #länge BY 1 DO
	                                                IF #gitter[#k].nummer > 0 THEN
	                                                    #gitter[#i].potenz_nummer[#gitter[#k].nummer - 1] := FALSE;
	                                                END_IF;
	                                            END_FOR;
	                                            IF #m < 2 THEN
	                                                #initial := #initial + 9;
	                                                #länge := #länge + 9;
	                                            END_IF;
	                                        END_FOR;
	                                    END_REGION
	                                    //Feldchen 80
	                                79:
	                                    REGION Feldchen 80
	                                        //Beschränkung mögliche Nummer in der Zeile 9
	                                        FOR #i := 72 TO 80 BY 1 DO
	                                            IF #gitter[#k].nummer > 0 THEN
	                                                #gitter[#i].potenz_nummer[#gitter[#k].nummer - 1] := FALSE;
	                                            END_IF;
	                                        END_FOR;
	                                        //Beschränkung mögliche Nummer in der Säule 8
	                                        FOR #i := 7 TO 80 BY 9 DO
	                                            IF #gitter[#k].nummer > 0 THEN
	                                                #gitter[#i].potenz_nummer[#gitter[#k].nummer - 1] := FALSE;
	                                            END_IF;
	                                        END_FOR;
	                                        //Beschränkung mögliche Nummer in dem Viereck 9
	                                        #initial := 60;
	                                        #länge := 62;
	                                        FOR #m := 0 TO 2 BY 1 DO
	                                            FOR #i := #initial TO #länge BY 1 DO
	                                                IF #gitter[#k].nummer > 0 THEN
	                                                    #gitter[#i].potenz_nummer[#gitter[#k].nummer - 1] := FALSE;
	                                                END_IF;
	                                            END_FOR;
	                                            IF #m < 2 THEN
	                                                #initial := #initial + 9;
	                                                #länge := #länge + 9;
	                                            END_IF;
	                                        END_FOR;
	                                    END_REGION
	                                    //Feldchen 81
	                                80:
	                                    REGION Feldchen 81
	                                        //Beschränkung mögliche Nummer in der Zeile 9
	                                        FOR #i := 72 TO 80 BY 1 DO
	                                            IF #gitter[#k].nummer > 0 THEN
	                                                #gitter[#i].potenz_nummer[#gitter[#k].nummer - 1] := FALSE;
	                                            END_IF;
	                                        END_FOR;
	                                        //Beschränkung mögliche Nummer in der Säule 9
	                                        FOR #i := 8 TO 80 BY 9 DO
	                                            IF #gitter[#k].nummer > 0 THEN
	                                                #gitter[#i].potenz_nummer[#gitter[#k].nummer - 1] := FALSE;
	                                            END_IF;
	                                        END_FOR;
	                                        //Beschränkung mögliche Nummer in dem Viereck 9
	                                        #initial := 60;
	                                        #länge := 62;
	                                        FOR #m := 0 TO 2 BY 1 DO
	                                            FOR #i := #initial TO #länge BY 1 DO
	                                                IF #gitter[#k].nummer > 0 THEN
	                                                    #gitter[#i].potenz_nummer[#gitter[#k].nummer - 1] := FALSE;
	                                                END_IF;
	                                            END_FOR;
	                                            IF #m < 2 THEN
	                                                #initial := #initial + 9;
	                                                #länge := #länge + 9;
	                                            END_IF;
	                                        END_FOR;
	                                    END_REGION
	                            END_CASE;
	                        END_REGION
	                    END_IF;
	                END_REGION
	                REGION Letze Nummer und Möglichkeiten Feld aufschreiben
	                    //Letze Nummer und Möglichkeiten Feld nach jeder Schleife aufschreiben
	                    FOR #i := 0 TO 80 BY 1 DO
	                        #gitter_letzte_num[#i].nummer := #gitter[#i].nummer;
	                        FOR #j := 0 TO 8 BY 1 DO
	                            #gitter_letzte_num[#i].potenz_nummer[#j] := #gitter[#i].potenz_nummer[#j];
	                        END_FOR;
	                    END_FOR;
	                END_REGION
	            END_FOR;
	        END_IF;
	    END_REGION
	END_REGION








END_FUNCTION_BLOCK

